# B&R Automation Studio project Lyskryds_i_to_retninger_jbl
Automation Studio 4.8.2.72

## Configuration Config1

### Hardware
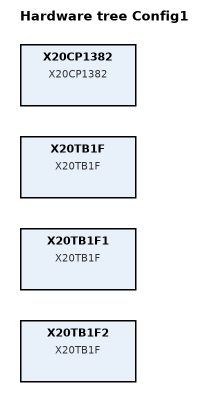
```
X20CP1382 : X20CP1382 v1.10.0.0  [X1 -> X1.SL; X2 -> X2.SL; X3 -> X3.SL]
  Module X1 (Type=X1, Virtual=true, Version=1.10.0.0)
    Connection (Connector=SS1, TargetModule=X20TB1F, TargetConnector=SS)
    Connection (Connector=SL, TargetModule=X20CP1382, TargetConnector=X1)
  Module X2 (Type=X2, Virtual=true, Version=1.10.0.0)
    Connection (Connector=SS1, TargetModule=X20TB1F1, TargetConnector=SS)
    Connection (Connector=SL, TargetModule=X20CP1382, TargetConnector=X2)
  Module X3 (Type=X3, Virtual=true, Version=1.10.0.0)
    Connection (Connector=SS1, TargetModule=X20TB1F2, TargetConnector=SS)
    Connection (Connector=SL, TargetModule=X20CP1382, TargetConnector=X3)
  Connector IF2:
    ActivateDevice = 1
  ConfigurationID = Lyskryds_i_to_retninger_jbl_Config1
  Simulation = 1
X20TB1F : X20TB1F v1.0.0.0
X20TB1F1 : X20TB1F v1.0.0.0
X20TB1F2 : X20TB1F v1.0.0.0
```

## Logical view

### Program Logical/Lyskryds (IEC)

#### Types.typ
```iecst
TYPE
	STOPPED_CASE :
		(
		a,
		b,
		c,
		d
		);
	TRAFFICLIGHT :
		(
		STOPPED,
		READY,
		STOP,
		GO
		);
END_TYPE
```

#### Variables.var
```iecst
VAR
	shift : BOOL;
	timer : TON;
	T1_state : TRAFFICLIGHT;
	T1_yellow : BOOL;
	T1_green : BOOL;
	T1_red : BOOL;
	T2_state : TRAFFICLIGHT;
	T2_yellow : BOOL;
	T2_green : BOOL;
	T2_red : BOOL;
	STOPPED_state : STOPPED_CASE;
END_VAR
```

#### Main.st
```iecst
(* NOTE: For mig har STOPPED_state ikke nogle værdi under watch medmindre man sletter den og sætter den ind i watch igen.
         Traffiklyset skifter som det skal selvom STOPPED_state ikke viser noget *)

PROGRAM _INIT
	// Define start states
	T1_state := GO;
	T2_state := STOPPED;
	STOPPED_state := a;
END_PROGRAM

PROGRAM _CYCLIC
	// Tilstandsskiftlogik / state change logic
	timer.IN := TRUE;
	CASE T1_state OF
		GO:
			timer.PT := T#2s;
			IF timer.Q AND shift THEN
				T1_state := STOP;
				timer.IN := FALSE;
			END_IF
			T2_state := STOPPED;

		STOP:
			timer.PT := T#2s;
			IF timer.Q THEN
				T1_state := STOPPED;
				timer.IN := FALSE;
			END_IF

		STOPPED:
			CASE STOPPED_state OF
				a:
					T2_state := READY;
					STOPPED_state := b;
				b:
					timer.PT := T#2s;
					IF timer.Q THEN
						T2_state := GO;
						timer.IN := FALSE;
						STOPPED_state := c;
					END_IF
				c:
					timer.PT := T#2s;
					IF T2_state = GO AND timer.Q AND shift THEN
						T2_state := STOP;
						timer.IN := FALSE;
						STOPPED_state := d;
					END_IF
				d:
					timer.PT := T#2s;
					IF timer.Q THEN
						T2_state := STOPPED;
						T1_state := READY;
						timer.IN := FALSE;
					END_IF
			END_CASE

		READY:
			STOPPED_state := a;
			timer.PT := T#2s;
			IF timer.Q THEN
				T1_state := GO;
				timer.IN := FALSE;
			END_IF
	END_CASE
	timer();

	// Trafficlight 1 - OUTPUT LOGIC
	CASE T1_state OF
		GO:
			T1_red := FALSE;
			T1_yellow := FALSE;
			T1_green := TRUE;
		STOP:
			T1_red := FALSE;
			T1_yellow := TRUE;
			T1_green := FALSE;
		STOPPED:
			T1_red := TRUE;
			T1_yellow := FALSE;
			T1_green := FALSE;
		READY:
			T1_red := TRUE;
			T1_yellow := TRUE;
			T1_green := FALSE;
	END_CASE

	// Trafficlight 2 - OUTPUT LOGIC
	CASE T2_state OF
		GO:
			T2_red := FALSE;
			T2_yellow := FALSE;
			T2_green := TRUE;
		STOP:
			T2_red := FALSE;
			T2_yellow := TRUE;
			T2_green := FALSE;
		STOPPED:
			T2_red := TRUE;
			T2_yellow := FALSE;
			T2_green := FALSE;
		READY:
			T2_red := TRUE;
			T2_yellow := TRUE;
			T2_green := FALSE;
	END_CASE
END_PROGRAM

PROGRAM _EXIT

END_PROGRAM
```

Listed in the project but not available here: Logical/Global.typ, Logical/Global.var, Logical/Libraries
